# EPICS substitutions: SM300/SM300-IOC-01App/Db/asyn_motor.substitutions
file $(MOTOR)/motorApp/Db/asyn_motor.db {

pattern {P,       N,     M,   DTYP,         PORT,       ADDR,        DESC,             EGU,  DIR,  VELO,  VBAS,  ACCL,  BDST,  BVEL,  BACC,  MRES,  PREC,  DHLM,  DLLM,  INIT}
        {"\$(P)", 1, "\$(M)", "asynMotor",  "\$(PORT)", "\$(ADDR)",  "\$(M) (SMC100)",  mm,  Pos,  1,     0,    .2,    0,     .5,     .2,    1,     0,     125,   -125,  ""}
}
